TEXTLIST PathChoice
  0 = 'Clockwise'
  1 = 'CounterClockwise'
   = ''
END_TEXTLIST

(* stored: Version 1.1.0.1
   TextList PathChoice: Id {5133fe1a-116b-47e4-96dc-5ff6e80ae6cb} *)
